FUNCTION_BLOCK TcoObjectTest EXTENDS TcoCore.TcoObject
VAR
	_MyIdentity				:	ULINT;
	_MyContextIdentity		:	ULINT;
	_MyContextStartCount 	:	ULINT;
	_MyContextEndCount		:	ULINT;
	_MyParentIdentity		:	ULINT;
	_TcoTaskTest_A			:	TcoTaskTest(THIS^);
	_TcoTaskTest_B			:	TcoTaskTest(THIS^);
	_TcoStateTest_A			:	TcoStateTest(THIS^, eRestoreMode.AutoRestoreMembers);
	_TcoStateTest_B			:	TcoStateTest(THIS^, eRestoreMode.None);
	// Object equality
	_TcoObjectEqualsTestObj1 	:   TcoObjectEqualsTest(THIS^);
	_TcoObjectEqualsTestObj2 	:   TcoObjectEqualsTest(THIS^);
END_VAR

{attribute 'TcRpcEnable'}
METHOD INTERNAL CallTaskInstancies
_TcoTaskTest_A();

_TcoTaskTest_B();
END_METHOD

{attribute 'TcRpcEnable'}
METHOD PUBLIC EqualsOverrideTest : BOOL
EqualsOverrideTest := _TcoObjectEqualsTestObj1.EqualsTo(_TcoObjectEqualsTestObj2);
END_METHOD

{attribute 'TcRpcEnable'}
METHOD PUBLIC EqualsTest : BOOL
VAR_INPUT
    _case : INT;
END_VAR

VAR
    referenceTo_a_TcoStateTest : REFERENCE TO TcoStateTest;
END_VAR
CASE _case OF
    0:
        referenceTo_a_TcoStateTest REF= _TcoStateTest_A;
        EqualsTest := _TcoStateTest_A.EqualsTo(referenceTo_a_TcoStateTest);
    1:
        EqualsTest := _TcoStateTest_A.EqualsTo(_TcoStateTest_B);
    4:
        EqualsTest := _TcoStateTest_B.EqualsTo(_TcoStateTest_A);
    2:
        EqualsTest := _TcoObjectEqualsTestObj1.EqualsTo(_TcoObjectEqualsTestObj1);
    3:
        EqualsTest := _TcoObjectEqualsTestObj1.EqualsTo(_TcoObjectEqualsTestObj2);
END_CASE
END_METHOD

{attribute 'TcRpcEnable'}
METHOD INTERNAL ReadOutIdentities
_MyIdentity			:=	THIS^.Identity;

_MyContextIdentity	:=	THIS^.Context.Identity;
		
_MyContextStartCount :=	THIS^.Context.StartCycleCount;

_MyContextEndCount	:=	THIS^.Context.EndCycleCount;

_MyParentIdentity	:=	THIS^._Parent.Identity;
END_METHOD

END_FUNCTION_BLOCK

(* stored: Version 1.1.0.1, ProductVersion 3.1.4024.6
   POU TcoObjectTest: Id {e84228ff-9c33-47a4-a38e-640688a82a88}, SpecialFunc None
   Method CallTaskInstancies: Id {ca9ba4d2-6103-4337-95bc-465f8f83317e}
   Method EqualsOverrideTest: Id {ee60d2fd-b5db-0d20-0c27-57a751cde2ce}
   Method EqualsTest: Id {9f06ff61-1678-0fe4-0121-54cfb8b16218}
   Method ReadOutIdentities: Id {b42bfa48-43e7-40ad-83bf-1125b1638f9d} *)
